// TIA Portal V18 export
FUNCTION_BLOCK "Pallet_Status"   // FB8, LAD
{ S7_Optimized_Access := 'TRUE' }
// stored: MemoryReserve 100, SetENOAutomatically false
   VAR_INPUT
      SensorA : Bool;
      SensorB : Bool;
      SensorC : Bool;
      SensorD : Bool;
   END_VAR
BEGIN
END_FUNCTION_BLOCK
